PROGRAM PRG_Task1
VAR
END_VAR

F_ConsumeTime(1000);

END_PROGRAM

(* stored: Version 1.1.0.1, ProductVersion 3.1.4026.18
   POU PRG_Task1: Id {a8d66589-a3a8-42eb-b177-33b0ce771de1}, SpecialFunc None *)
